FUNCTION_BLOCK fbDigitalInput EXTENDS fbDigitalIO

END_FUNCTION_BLOCK

(* stored: Version 1.1.0.1, ProductVersion 3.1.4024.15
   POU fbDigitalInput: Id {cb513b1f-4e9c-4f9b-9fec-6b5dbb71decd}, SpecialFunc None *)
